FUNCTION_BLOCK FB_TelescopeSlewingState EXTENDS FB_TelescopeState
VAR_INPUT
END_VAR
VAR_OUTPUT
END_VAR
VAR
	pMachine : POINTER TO FB_TelescopeMachine;
END_VAR

METHOD FB_init : BOOL
VAR_INPUT
	bInitRetains : BOOL; // if TRUE, the retain variables are initialized (warm start / cold start)
	bInCopyCode : BOOL;  // if TRUE, the instance afterwards gets moved into the copy code (online change)
	pMachine : POINTER TO FB_TelescopeMachine;
END_VAR
THIS^.pMachine := pMachine;
END_METHOD

METHOD Park : BOOL
VAR_INPUT
END_VAR
END_METHOD

METHOD Slew : BOOL
VAR_INPUT
	fAzimuth	: LREAL;
	fAltitude	: LREAL;
END_VAR
END_METHOD

METHOD Stop : BOOL
VAR_INPUT
END_VAR
END_METHOD

METHOD Track : BOOL
VAR_INPUT
	fRightAscension	: LREAL;
	fDeclination	: LREAL;
END_VAR
END_METHOD

END_FUNCTION_BLOCK

(* stored: Version 1.1.0.1, ProductVersion 3.1.4024.15
   POU FB_TelescopeSlewingState: Id {edf837d7-00f7-4665-86d4-0431da6cffec}, SpecialFunc None
   Method FB_init: Id {7b51a5dc-97b4-45ed-9e5c-4aa95e9a2bef}
   Method Park: Id {b917d2c7-d098-4540-9842-edfdeaaf0bcd}
   Method Slew: Id {0f710bfe-2197-4b37-849c-9bf1417623c0}
   Method Stop: Id {e027a8c8-3486-40d1-a1fe-d2068ce4d75f}
   Method Track: Id {e3d5ebbe-9256-4180-9dd6-2ad33d746f90} *)
